// LS Electric XG5000 project: 8_28
// PLC LSPLC
// module base 0 slot 0: 입출력 모듈:XBC-DR14E (DC 24V 입력 8점, 릴레이 출력 6점)

PROGRAM NewProgram (task: 스캔 프로그램)

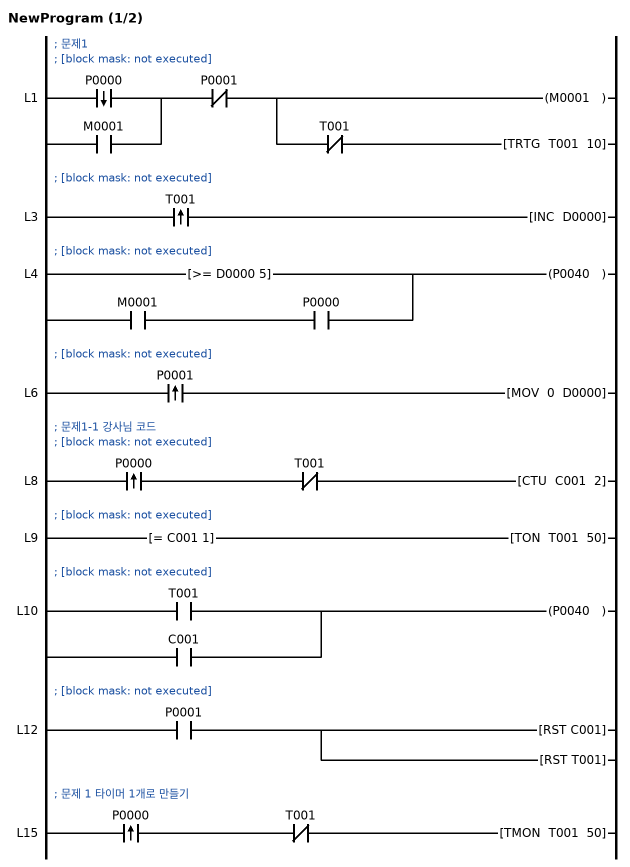
// 문제1
; L1 (block mask: not executed)
LOADN     P0000
OR        M0001
AND NOT   P0001
OUT       M0001
AND NOT   T001
TRTG      T001 10
; L3 (block mask: not executed)
LOADP     T001
INC       D0000
; L4 (block mask: not executed)
LOAD>=    D0000 5
LOAD      M0001
AND       P0000
OR LOAD
OUT       P0040
; L6 (block mask: not executed)
LOADP     P0001
MOV       0 D0000
// 문제1-1 강사님 코드
; L8 (block mask: not executed)
LOADP     P0000
AND NOT   T001
CTU       C001 2
; L9 (block mask: not executed)
LOAD=     C001 1
TON       T001 50
; L10 (block mask: not executed)
LOAD      T001
OR        C001
OUT       P0040
; L12 (block mask: not executed)
LOAD      P0001
RST       C001
RST       T001
// 문제 1 타이머 1개로 만들기
; L15
LOADP     P0000
AND NOT   T001
TMON      T001 50

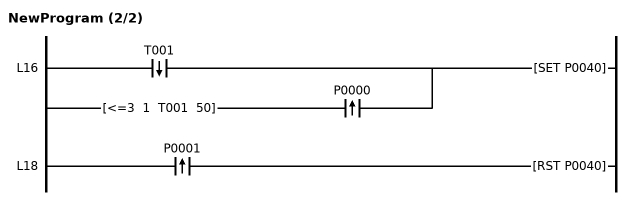
; L16
LOADN     T001
LOAD<=3   1 T001 50
ANDP      P0000
OR LOAD
SET       P0040
; L18
LOADP     P0001
RST       P0040